(* PLC project model, Beckhoff Automation Beckhoff MLlib 3.1.251201.0 *)
(* stored: creationDateTime 2026-07-10T12:15:09.7362232, modificationDateTime 2026-07-10T12:15:09.7362232 *)

TYPE ST_modelInput :
STRUCT

	{attribute 'hide'} _header_DO_NOT_CHANGE : ARRAY[0..63] OF SINT := [-1,-112,120,86,52,18,-1,-1,1,-1,0,0,-1,-1,-112,-112,65,64,108,85,118,21,-37,1,110,122,-102,19,93,-117,-35,-43,3,-45,33,-52,25,-24,90,7,83,36,22,5,-43,-65,-103,-61,76,0,0,0,0,0,0,0,0,0,0,0,0,0,0,0];
	in_float_input : ARRAY[0..0,0..2] OF REAL;

END_STRUCT
END_TYPE

TYPE ST_modelOutput :
STRUCT

	{attribute 'hide'} _header_DO_NOT_CHANGE : ARRAY[0..63] OF SINT := [-1,-112,120,86,52,18,-1,-1,1,-1,0,0,-1,-1,-112,-112,-35,24,-50,75,-65,96,-121,123,127,87,61,127,-39,-108,16,-70,120,-89,-28,78,-43,26,-32,-7,81,19,29,-89,-55,3,43,2,68,0,0,0,0,0,0,0,0,0,0,0,0,0,0,0];
	out_variable : ARRAY[0..0,0..0] OF REAL;

END_STRUCT
END_TYPE
